// TwinCAT 3 PLC project EIOSM000003
// ProgramVersion: 3.1.4024.0
// libraries:
//   EfficientIO Communicator, * (EfficientIO)
//   EfficientIO Energy Basic, * (EfficientIO)
//   Lynus Persistent Data V1, * (Lynus AG)
//   Lynus Standards, * (EfficientIO)
//   Tc2_EtherCAT, * (Beckhoff Automation GmbH)
//   Tc2_Standard, * (Beckhoff Automation GmbH)
//   Tc2_System, * (Beckhoff Automation GmbH)
//   Tc2_Utilities, * (Beckhoff Automation GmbH)
//   Tc3_IPCDiag, * (Beckhoff Automation GmbH)
//   Tc3_Module, * (Beckhoff Automation GmbH)
// project tree:
//   ENUM/ E_State.TcDUT (not stored)
//   / FastTask.TcTTO, PlcTask.TcTTO, SlowTask.TcTTO
//   FBs/EL3443_DPM/DUTs/ E_EL3443_DPM_Phase.TcDUT (not stored), E_EL3443_DPM_Total.TcDUT (not stored), MDP5001_341_7CD731EE.TcDUT (not stored), MDP5001_341_I_7CD731EE.TcDUT (not stored), MDP5001_341_O_7CD731EE.TcDUT (not stored), ST_EL3443_DPM_MUX_REAL.TcDUT (not stored), ST_EL3443_DPM_MUX_ULINT.TcDUT (not stored), ST_EL3443_DPM_StatusLx.TcDUT (not stored), ST_EL3443_DPM_StatusTotal.TcDUT (not stored), ST_EL3443_DPM_VariantLx.TcDUT (not stored), ST_EL3443_DPM_VariantTotal.TcDUT (not stored), ST_EL3443_DPM_VariantValues.TcDUT (not stored)
//   FBs/EL3443_DPM/ FB_EL3443_DPM.TcPOU (not stored)
//   FBs/EL3446 FW02 or higher/DUTs/ E_EL3446_Phase.TcDUT (not stored), MDP5001_342_066CA8C6.TcDUT (not stored), MDP5001_342_I_066CA8C6.TcDUT (not stored), MDP5001_342_O_066CA8C6.TcDUT (not stored), ST_EL3446_MUX_REAL.TcDUT (not stored), ST_EL3446_MUX_ULINT.TcDUT (not stored), ST_EL3446_StatusIx.TcDUT (not stored), ST_EL3446_VariantIx.TcDUT (not stored), ST_EL3446_VariantValues.TcDUT (not stored)
//   FBs/EL3446 FW02 or higher/ FB_EL3446.TcPOU (not stored)
//   FBs/ FB_CoE_EL3443.TcPOU (not stored), FB_CoE_EL3446.TcPOU (not stored), FB_EM_Beckhoff_EL3443.TcPOU (not stored), FB_EM_Beckhoff_EL3446.TcPOU (not stored), FB_PT100_Read.TcPOU, prg_ReadDeviceName.TcPOU (not stored)
//   POUs/ prgComEffIO.TcPOU, prgEM.TcPOU, prgHW.TcPOU (not stored), prgPersistent.TcPOU (not stored), prgRWEffIO.TcPOU (not stored), prgTmp.TcPOU, prgVarEffIO.TcPOU (not stored)
// real-time tasks:
//   TASK MiddleTask: cycle T#10ms, priority 20, ADS port 350
//   TASK FastTask: cycle T#5ms, priority 19, ADS port 351
//   TASK SlowTask: cycle T#20ms, priority 21, ADS port 352
// I/O:
//   DEVICE Device 1 (Beckhoff CCAT)
//   DEVICE Device 2 (EtherCAT), AmsNetId 5.146.122.92.3.1
//     Term 1 (EK1200) [EK1200-5000 EtherCAT Power supply (2A E-Bus)]
//       Term 2 (EL3443) [EL3443 3Ch. Power Measuring]
//       Term 3 (EL3446) [EL3446 6 Ch.DPM Current Measurement Terminal]
//       Term 4 (EL3446) [EL3446 6 Ch.DPM Current Measurement Terminal]
//       Term 5 (EL3446) [EL3446 6 Ch.DPM Current Measurement Terminal]
//       Term 6 (EL3446) [EL3446 6 Ch.DPM Current Measurement Terminal]
//       Term 7 (EL3202) [EL3202 2Ch. Ana. Input PT100 (RTD)]
//       Term 8 (EL9011) [EL9011 End Terminal]
// variable links:
//   EIOSM000003/EIOSM000003 Instance <-> Device 2 (EtherCAT)/Term 1 (EK1200)/Term 2 (EL3443)
//     PlcTask Inputs/prgHW.MDP5001_341_DPM_Data_Data_{1..20} <-> DPM Data/Data {1..20}  (20 links)
//     PlcTask Inputs/prgHW.MDP5001_341_L1_Basic_Current <-> L1 Basic/Current
//     PlcTask Inputs/prgHW.MDP5001_341_L2_Basic_Current <-> L2 Basic/Current
//     PlcTask Inputs/prgHW.MDP5001_341_L3_Basic_Current <-> L3 Basic/Current
//     PlcTask Inputs/prgHW.MDP5001_341_L1_Basic_Voltage <-> L1 Basic/Voltage
//     PlcTask Inputs/prgHW.MDP5001_341_L2_Basic_Voltage <-> L2 Basic/Voltage
//     PlcTask Inputs/prgHW.MDP5001_341_L3_Basic_Voltage <-> L3 Basic/Voltage
//     PlcTask Inputs/prgHW.MDP5001_341_L1_Power_Active_Power <-> L1 Power/Active Power
//     PlcTask Inputs/prgHW.MDP5001_341_L2_Power_Active_Power <-> L2 Power/Active Power
//     PlcTask Inputs/prgHW.MDP5001_341_L3_Power_Active_Power <-> L3 Power/Active Power
//     PlcTask Inputs/prgHW.MDP5001_341_L1_Power_Apparent_Power <-> L1 Power/Apparent Power
//     PlcTask Inputs/prgHW.MDP5001_341_L2_Power_Apparent_Power <-> L2 Power/Apparent Power
//     PlcTask Inputs/prgHW.MDP5001_341_L3_Power_Apparent_Power <-> L3 Power/Apparent Power
//     PlcTask Inputs/prgHW.MDP5001_341_L1_Power_Power_Factor <-> L1 Power/Power Factor
//     PlcTask Inputs/prgHW.MDP5001_341_L2_Power_Power_Factor <-> L2 Power/Power Factor
//     PlcTask Inputs/prgHW.MDP5001_341_L3_Power_Power_Factor <-> L3 Power/Power Factor
//     PlcTask Inputs/prgHW.MDP5001_341_L1_Power_Reactive_Power <-> L1 Power/Reactive Power
//     PlcTask Inputs/prgHW.MDP5001_341_L2_Power_Reactive_Power <-> L2 Power/Reactive Power
//     PlcTask Inputs/prgHW.MDP5001_341_L3_Power_Reactive_Power <-> L3 Power/Reactive Power
//     PlcTask Inputs/prgHW.MDP5001_341_L1_Status_Current_Guard_Error <-> L1 Status/Current Guard Error
//     PlcTask Inputs/prgHW.MDP5001_341_L2_Status_Current_Guard_Error <-> L2 Status/Current Guard Error
//     PlcTask Inputs/prgHW.MDP5001_341_L3_Status_Current_Guard_Error <-> L3 Status/Current Guard Error
//     PlcTask Inputs/prgHW.MDP5001_341_L1_Status_Current_Guard_Warning <-> L1 Status/Current Guard Warning
//     PlcTask Inputs/prgHW.MDP5001_341_L2_Status_Current_Guard_Warning <-> L2 Status/Current Guard Warning
//     PlcTask Inputs/prgHW.MDP5001_341_L3_Status_Current_Guard_Warning <-> L3 Status/Current Guard Warning
//     PlcTask Inputs/prgHW.MDP5001_341_L1_Status_Inaccurate_Current <-> L1 Status/Inaccurate Current
//     PlcTask Inputs/prgHW.MDP5001_341_L2_Status_Inaccurate_Current <-> L2 Status/Inaccurate Current
//     PlcTask Inputs/prgHW.MDP5001_341_L3_Status_Inaccurate_Current <-> L3 Status/Inaccurate Current
//     PlcTask Inputs/prgHW.MDP5001_341_L1_Status_Inaccurate_Voltage <-> L1 Status/Inaccurate Voltage
//     PlcTask Inputs/prgHW.MDP5001_341_L2_Status_Inaccurate_Voltage <-> L2 Status/Inaccurate Voltage
//     PlcTask Inputs/prgHW.MDP5001_341_L3_Status_Inaccurate_Voltage <-> L3 Status/Inaccurate Voltage
//     PlcTask Inputs/prgHW.MDP5001_341_L1_Status_Overcurrent <-> L1 Status/Overcurrent
//     PlcTask Inputs/prgHW.MDP5001_341_L2_Status_Overcurrent <-> L2 Status/Overcurrent
//     PlcTask Inputs/prgHW.MDP5001_341_L3_Status_Overcurrent <-> L3 Status/Overcurrent
//     PlcTask Inputs/prgHW.MDP5001_341_L1_Status_Overvoltage <-> L1 Status/Overvoltage
//     PlcTask Inputs/prgHW.MDP5001_341_L2_Status_Overvoltage <-> L2 Status/Overvoltage
//     PlcTask Inputs/prgHW.MDP5001_341_L3_Status_Overvoltage <-> L3 Status/Overvoltage
//     PlcTask Inputs/prgHW.MDP5001_341_L1_Status_TxPDO_Toggle <-> L1 Status/TxPDO Toggle
//     PlcTask Inputs/prgHW.MDP5001_341_L2_Status_TxPDO_Toggle <-> L2 Status/TxPDO Toggle
//     PlcTask Inputs/prgHW.MDP5001_341_L3_Status_TxPDO_Toggle <-> L3 Status/TxPDO Toggle
//     PlcTask Inputs/prgHW.MDP5001_341_L1_Status_Voltage_Guard_Error <-> L1 Status/Voltage Guard Error
//     PlcTask Inputs/prgHW.MDP5001_341_L2_Status_Voltage_Guard_Error <-> L2 Status/Voltage Guard Error
//     PlcTask Inputs/prgHW.MDP5001_341_L3_Status_Voltage_Guard_Error <-> L3 Status/Voltage Guard Error
//     PlcTask Inputs/prgHW.MDP5001_341_L1_Status_Voltage_Guard_Warning <-> L1 Status/Voltage Guard Warning
//     PlcTask Inputs/prgHW.MDP5001_341_L2_Status_Voltage_Guard_Warning <-> L2 Status/Voltage Guard Warning
//     PlcTask Inputs/prgHW.MDP5001_341_L3_Status_Voltage_Guard_Warning <-> L3 Status/Voltage Guard Warning
//     PlcTask Inputs/prgHW.MDP5001_341_L1_Status_Voltage_Sign_Bit <-> L1 Status/Voltage Sign Bit
//     PlcTask Inputs/prgHW.MDP5001_341_L2_Status_Voltage_Sign_Bit <-> L2 Status/Voltage Sign Bit
//     PlcTask Inputs/prgHW.MDP5001_341_L3_Status_Voltage_Sign_Bit <-> L3 Status/Voltage Sign Bit
//     PlcTask Inputs/prgHW.MDP5001_341_Total_Basic_Calculated_Neutral_Line_Current <-> Total Basic/Calculated Neutral Line Current
//     PlcTask Inputs/prgHW.MDP5001_341_Total_Basic_Frequency <-> Total Basic/Frequency
//     PlcTask Inputs/prgHW.MDP5001_341_Total_Basic_Power_Factor <-> Total Basic/Power Factor
//     PlcTask Inputs/prgHW.MDP5001_341_Total_Status_Active_Power_Guard_Error <-> Total Status/Active Power Guard Error
//     PlcTask Inputs/prgHW.MDP5001_341_Total_Status_Active_Power_Guard_Warning <-> Total Status/Active Power Guard Warning
//     PlcTask Inputs/prgHW.MDP5001_341_Total_Status_Apparent_Power_Guard_Error <-> Total Status/Apparent Power Guard Error
//     PlcTask Inputs/prgHW.MDP5001_341_Total_Status_Apparent_Power_Guard_Warning <-> Total Status/Apparent Power Guard Warning
//     PlcTask Inputs/prgHW.MDP5001_341_Total_Status_Frequency_Guard_Error <-> Total Status/Frequency Guard Error
//     PlcTask Inputs/prgHW.MDP5001_341_Total_Status_Frequency_Guard_Warning <-> Total Status/Frequency Guard Warning
//     PlcTask Inputs/prgHW.MDP5001_341_Total_Status_Grid_Direction <-> Total Status/Grid Direction
//     PlcTask Inputs/prgHW.MDP5001_341_Total_Status_Neutral_Current_Guard_Error <-> Total Status/Neutral Current Guard Error
//     PlcTask Inputs/prgHW.MDP5001_341_Total_Status_Neutral_Current_Guard_Warning <-> Total Status/Neutral Current Guard Warning
//     PlcTask Inputs/prgHW.MDP5001_341_Total_Status_Power_Quality_Factor <-> Total Status/Power Quality Factor
//     PlcTask Inputs/prgHW.MDP5001_341_Total_Status_Power_Quality_Guard_Error <-> Total Status/Power Quality Guard Error
//     PlcTask Inputs/prgHW.MDP5001_341_Total_Status_Power_Quality_Guard_Warning <-> Total Status/Power Quality Guard Warning
//     PlcTask Inputs/prgHW.MDP5001_341_Total_Status_System_State <-> Total Status/System State
//     PlcTask Inputs/prgHW.MDP5001_341_Total_Status_TxPDO_State <-> Total Status/TxPDO State
//     PlcTask Inputs/prgHW.MDP5001_341_Total_Status_TxPDO_Toggle <-> Total Status/TxPDO Toggle
//     PlcTask Inputs/prgHW.MDP5001_341_Total_Variant_Value_In_Index_1_REAL <-> Total Variant Value In/Index 1 REAL
//     PlcTask Inputs/prgHW.MDP5001_341_Total_Variant_Value_In_Index_2_REAL <-> Total Variant Value In/Index 2 REAL
//     PlcTask Inputs/prgHW.MDP5001_341_Total_Variant_Value_In_Index_3_REAL <-> Total Variant Value In/Index 3 REAL
//     PlcTask Inputs/prgHW.MDP5001_341_Total_Variant_Value_In_Index_4_ULINT <-> Total Variant Value In/Index 4 ULINT
//     PlcTask Inputs/prgHW.MDP5001_341_Total_Variant_Value_In_TxPDO_Toggle <-> Total Variant Value In/TxPDO Toggle
//     PlcTask Inputs/prgHW.MDP5001_341_Total_Variant_Value_In_Value_1_REAL <-> Total Variant Value In/Value 1 REAL
//     PlcTask Inputs/prgHW.MDP5001_341_Total_Variant_Value_In_Value_2_REAL <-> Total Variant Value In/Value 2 REAL
//     PlcTask Inputs/prgHW.MDP5001_341_Total_Variant_Value_In_Value_3_REAL <-> Total Variant Value In/Value 3 REAL
//     PlcTask Inputs/prgHW.MDP5001_341_Total_Variant_Value_In_Value_4_ULINT <-> Total Variant Value In/Value 4 ULINT
//     PlcTask Outputs/prgHW.MDP5001_341_Total_Interval_Reset_Interval <-> Total Interval/Reset Interval
//     PlcTask Outputs/prgHW.MDP5001_341_Total_Variant_Value_Out_Index_1_REAL <-> Total Variant Value Out/Index 1 REAL
//     PlcTask Outputs/prgHW.MDP5001_341_Total_Variant_Value_Out_Index_2_REAL <-> Total Variant Value Out/Index 2 REAL
//     PlcTask Outputs/prgHW.MDP5001_341_Total_Variant_Value_Out_Index_3_REAL <-> Total Variant Value Out/Index 3 REAL
//     PlcTask Outputs/prgHW.MDP5001_341_Total_Variant_Value_Out_Index_4_ULINT <-> Total Variant Value Out/Index 4 ULINT
//   EIOSM000003/EIOSM000003 Instance <-> Device 2 (EtherCAT)/Term 1 (EK1200)/Term 3 (EL3446)
//     PlcTask Inputs/prgHW.MDP5001_342_DPM_Variant_Value_In_Index_1_REAL_EM1 <-> DPM Variant Value In/Index 1 REAL
//     PlcTask Inputs/prgHW.MDP5001_342_DPM_Variant_Value_In_Index_2_REAL_EM1 <-> DPM Variant Value In/Index 2 REAL
//     PlcTask Inputs/prgHW.MDP5001_342_DPM_Variant_Value_In_Index_3_REAL_EM1 <-> DPM Variant Value In/Index 3 REAL
//     PlcTask Inputs/prgHW.MDP5001_342_DPM_Variant_Value_In_Index_4_ULINT_EM1 <-> DPM Variant Value In/Index 4 ULINT
//     PlcTask Inputs/prgHW.MDP5001_342_DPM_Variant_Value_In_TxPDO_Toggle_EM1 <-> DPM Variant Value In/TxPDO Toggle
//     PlcTask Inputs/prgHW.MDP5001_342_DPM_Variant_Value_In_Value_1_REAL_EM1 <-> DPM Variant Value In/Value 1 REAL
//     PlcTask Inputs/prgHW.MDP5001_342_DPM_Variant_Value_In_Value_2_REAL_EM1 <-> DPM Variant Value In/Value 2 REAL
//     PlcTask Inputs/prgHW.MDP5001_342_DPM_Variant_Value_In_Value_3_REAL_EM1 <-> DPM Variant Value In/Value 3 REAL
//     PlcTask Inputs/prgHW.MDP5001_342_DPM_Variant_Value_In_Value_4_ULINT_EM1 <-> DPM Variant Value In/Value 4 ULINT
//     PlcTask Inputs/prgHW.MDP5001_342_I{1..6}_Channel_Active_Energy_EM1 <-> I{1..6} Channel/Active Energy  (6 links)
//     PlcTask Inputs/prgHW.MDP5001_342_I{1..6}_Channel_Active_Power_EM1 <-> I{1..6} Channel/Active Power  (6 links)
//     PlcTask Inputs/prgHW.MDP5001_342_I{1..6}_Channel_Active_Power_Guard_Error_EM1 <-> I{1..6} Channel/Active Power Guard Error  (6 links)
//     PlcTask Inputs/prgHW.MDP5001_342_I{1..6}_Channel_Active_Power_Guard_Warning_EM1 <-> I{1..6} Channel/Active Power Guard Warning  (6 links)
//     PlcTask Inputs/prgHW.MDP5001_342_I{1..6}_Channel_Apparent_Power_EM1 <-> I{1..6} Channel/Apparent Power  (6 links)
//     PlcTask Inputs/prgHW.MDP5001_342_I{1..6}_Channel_Apparent_Power_Guard_Error_EM1 <-> I{1..6} Channel/Apparent Power Guard Error  (6 links)
//     PlcTask Inputs/prgHW.MDP5001_342_I{1..6}_Channel_Apparent_Power_Guard_Warning_EM1 <-> I{1..6} Channel/Apparent Power Guard Warning  (6 links)
//     PlcTask Inputs/prgHW.MDP5001_342_I{1..6}_Channel_Current_EM1 <-> I{1..6} Channel/Current  (6 links)
//     PlcTask Inputs/prgHW.MDP5001_342_I{1..6}_Channel_Current_Guard_Error_EM1 <-> I{1..6} Channel/Current Guard Error  (6 links)
//     PlcTask Inputs/prgHW.MDP5001_342_I{1..6}_Channel_Current_Guard_Warning_EM1 <-> I{1..6} Channel/Current Guard Warning  (6 links)
//     PlcTask Inputs/prgHW.MDP5001_342_I{1..6}_Channel_DPM_Inaccurate_EM1 <-> I{1..6} Channel/DPM Inaccurate  (6 links)
//     PlcTask Inputs/prgHW.MDP5001_342_I{1..6}_Channel_DPM_Timeout_EM1 <-> I{1..6} Channel/DPM Timeout  (6 links)
//     PlcTask Inputs/prgHW.MDP5001_342_I{1..6}_Channel_Inaccurate_Current_EM1 <-> I{1..6} Channel/Inaccurate Current  (6 links)
//     PlcTask Inputs/prgHW.MDP5001_342_I{1..6}_Channel_Overcurrent_EM1 <-> I{1..6} Channel/Overcurrent  (6 links)
//     PlcTask Inputs/prgHW.MDP5001_342_I{1..6}_Channel_Reactive_Power_Fundamental_EM1 <-> I{1..6} Channel/Reactive Power Fundamental  (6 links)
//     PlcTask Inputs/prgHW.MDP5001_342_I{1..6}_Channel_Reactive_Power_Guard_Error_EM1 <-> I{1..6} Channel/Reactive Power Guard Error  (6 links)
//     PlcTask Inputs/prgHW.MDP5001_342_I{1..6}_Channel_Reactive_Power_Guard_Warning_EM1 <-> I{1..6} Channel/Reactive Power Guard Warning  (6 links)
//     PlcTask Inputs/prgHW.MDP5001_342_I{1..6}_Channel_TxPDO_Toggle_EM1 <-> I{1..6} Channel/TxPDO Toggle  (6 links)
//     PlcTask Outputs/prgHW.MDP5001_342_DPM_Data_Data_{1..20}_EM1 <-> DPM Data/Data {1..20}  (20 links)
//     PlcTask Outputs/prgHW.MDP5001_342_DPM_Variant_Value_Out_Index_1_REAL_EM1 <-> DPM Variant Value Out/Index 1 REAL
//     PlcTask Outputs/prgHW.MDP5001_342_DPM_Variant_Value_Out_Index_2_REAL_EM1 <-> DPM Variant Value Out/Index 2 REAL
//     PlcTask Outputs/prgHW.MDP5001_342_DPM_Variant_Value_Out_Index_3_REAL_EM1 <-> DPM Variant Value Out/Index 3 REAL
//     PlcTask Outputs/prgHW.MDP5001_342_DPM_Variant_Value_Out_Index_4_ULINT_EM1 <-> DPM Variant Value Out/Index 4 ULINT
//   EIOSM000003/EIOSM000003 Instance <-> Device 2 (EtherCAT)/Term 1 (EK1200)/Term 4 (EL3446)
//     PlcTask Inputs/prgHW.MDP5001_342_DPM_Variant_Value_In_Index_1_REAL_EM2 <-> DPM Variant Value In/Index 1 REAL
//     PlcTask Inputs/prgHW.MDP5001_342_DPM_Variant_Value_In_Index_2_REAL_EM2 <-> DPM Variant Value In/Index 2 REAL
//     PlcTask Inputs/prgHW.MDP5001_342_DPM_Variant_Value_In_Index_3_REAL_EM2 <-> DPM Variant Value In/Index 3 REAL
//     PlcTask Inputs/prgHW.MDP5001_342_DPM_Variant_Value_In_Index_4_ULINT_EM2 <-> DPM Variant Value In/Index 4 ULINT
//     PlcTask Inputs/prgHW.MDP5001_342_DPM_Variant_Value_In_TxPDO_Toggle_EM2 <-> DPM Variant Value In/TxPDO Toggle
//     PlcTask Inputs/prgHW.MDP5001_342_DPM_Variant_Value_In_Value_1_REAL_EM2 <-> DPM Variant Value In/Value 1 REAL
//     PlcTask Inputs/prgHW.MDP5001_342_DPM_Variant_Value_In_Value_2_REAL_EM2 <-> DPM Variant Value In/Value 2 REAL
//     PlcTask Inputs/prgHW.MDP5001_342_DPM_Variant_Value_In_Value_3_REAL_EM2 <-> DPM Variant Value In/Value 3 REAL
//     PlcTask Inputs/prgHW.MDP5001_342_DPM_Variant_Value_In_Value_4_ULINT_EM2 <-> DPM Variant Value In/Value 4 ULINT
//     PlcTask Inputs/prgHW.MDP5001_342_I{1..6}_Channel_Active_Energy_EM2 <-> I{1..6} Channel/Active Energy  (6 links)
//     PlcTask Inputs/prgHW.MDP5001_342_I{1..6}_Channel_Active_Power_EM2 <-> I{1..6} Channel/Active Power  (6 links)
//     PlcTask Inputs/prgHW.MDP5001_342_I{1..6}_Channel_Active_Power_Guard_Error_EM2 <-> I{1..6} Channel/Active Power Guard Error  (6 links)
//     PlcTask Inputs/prgHW.MDP5001_342_I{1..6}_Channel_Active_Power_Guard_Warning_EM2 <-> I{1..6} Channel/Active Power Guard Warning  (6 links)
//     PlcTask Inputs/prgHW.MDP5001_342_I{1..6}_Channel_Apparent_Power_EM2 <-> I{1..6} Channel/Apparent Power  (6 links)
//     PlcTask Inputs/prgHW.MDP5001_342_I{1..6}_Channel_Apparent_Power_Guard_Error_EM2 <-> I{1..6} Channel/Apparent Power Guard Error  (6 links)
//     PlcTask Inputs/prgHW.MDP5001_342_I{1..6}_Channel_Apparent_Power_Guard_Warning_EM2 <-> I{1..6} Channel/Apparent Power Guard Warning  (6 links)
//     PlcTask Inputs/prgHW.MDP5001_342_I{1..6}_Channel_Current_EM2 <-> I{1..6} Channel/Current  (6 links)
//     PlcTask Inputs/prgHW.MDP5001_342_I{1..6}_Channel_Current_Guard_Error_EM2 <-> I{1..6} Channel/Current Guard Error  (6 links)
//     PlcTask Inputs/prgHW.MDP5001_342_I{1..6}_Channel_Current_Guard_Warning_EM2 <-> I{1..6} Channel/Current Guard Warning  (6 links)
//     PlcTask Inputs/prgHW.MDP5001_342_I{1..6}_Channel_DPM_Inaccurate_EM2 <-> I{1..6} Channel/DPM Inaccurate  (6 links)
//     PlcTask Inputs/prgHW.MDP5001_342_I{1..6}_Channel_DPM_Timeout_EM2 <-> I{1..6} Channel/DPM Timeout  (6 links)
//     PlcTask Inputs/prgHW.MDP5001_342_I{1..6}_Channel_Inaccurate_Current_EM2 <-> I{1..6} Channel/Inaccurate Current  (6 links)
//     PlcTask Inputs/prgHW.MDP5001_342_I{1..6}_Channel_Overcurrent_EM2 <-> I{1..6} Channel/Overcurrent  (6 links)
//     PlcTask Inputs/prgHW.MDP5001_342_I{1..6}_Channel_Reactive_Power_Fundamental_EM2 <-> I{1..6} Channel/Reactive Power Fundamental  (6 links)
//     PlcTask Inputs/prgHW.MDP5001_342_I{1..6}_Channel_Reactive_Power_Guard_Error_EM2 <-> I{1..6} Channel/Reactive Power Guard Error  (6 links)
//     PlcTask Inputs/prgHW.MDP5001_342_I{1..6}_Channel_Reactive_Power_Guard_Warning_EM2 <-> I{1..6} Channel/Reactive Power Guard Warning  (6 links)
//     PlcTask Inputs/prgHW.MDP5001_342_I{1..6}_Channel_TxPDO_Toggle_EM2 <-> I{1..6} Channel/TxPDO Toggle  (6 links)
//     PlcTask Outputs/prgHW.MDP5001_342_DPM_Data_Data_{1..20}_EM2 <-> DPM Data/Data {1..20}  (20 links)
//     PlcTask Outputs/prgHW.MDP5001_342_DPM_Variant_Value_Out_Index_1_REAL_EM2 <-> DPM Variant Value Out/Index 1 REAL
//     PlcTask Outputs/prgHW.MDP5001_342_DPM_Variant_Value_Out_Index_2_REAL_EM2 <-> DPM Variant Value Out/Index 2 REAL
//     PlcTask Outputs/prgHW.MDP5001_342_DPM_Variant_Value_Out_Index_3_REAL_EM2 <-> DPM Variant Value Out/Index 3 REAL
//     PlcTask Outputs/prgHW.MDP5001_342_DPM_Variant_Value_Out_Index_4_ULINT_EM2 <-> DPM Variant Value Out/Index 4 ULINT
//   EIOSM000003/EIOSM000003 Instance <-> Device 2 (EtherCAT)/Term 1 (EK1200)/Term 5 (EL3446)
//     PlcTask Inputs/prgHW.MDP5001_342_DPM_Variant_Value_In_Index_1_REAL_EM3 <-> DPM Variant Value In/Index 1 REAL
//     PlcTask Inputs/prgHW.MDP5001_342_DPM_Variant_Value_In_Index_2_REAL_EM3 <-> DPM Variant Value In/Index 2 REAL
//     PlcTask Inputs/prgHW.MDP5001_342_DPM_Variant_Value_In_Index_3_REAL_EM3 <-> DPM Variant Value In/Index 3 REAL
//     PlcTask Inputs/prgHW.MDP5001_342_DPM_Variant_Value_In_Index_4_ULINT_EM3 <-> DPM Variant Value In/Index 4 ULINT
//     PlcTask Inputs/prgHW.MDP5001_342_DPM_Variant_Value_In_TxPDO_Toggle_EM3 <-> DPM Variant Value In/TxPDO Toggle
//     PlcTask Inputs/prgHW.MDP5001_342_DPM_Variant_Value_In_Value_1_REAL_EM3 <-> DPM Variant Value In/Value 1 REAL
//     PlcTask Inputs/prgHW.MDP5001_342_DPM_Variant_Value_In_Value_2_REAL_EM3 <-> DPM Variant Value In/Value 2 REAL
//     PlcTask Inputs/prgHW.MDP5001_342_DPM_Variant_Value_In_Value_3_REAL_EM3 <-> DPM Variant Value In/Value 3 REAL
//     PlcTask Inputs/prgHW.MDP5001_342_DPM_Variant_Value_In_Value_4_ULINT_EM3 <-> DPM Variant Value In/Value 4 ULINT
//     PlcTask Inputs/prgHW.MDP5001_342_I{1..6}_Channel_Active_Energy_EM3 <-> I{1..6} Channel/Active Energy  (6 links)
//     PlcTask Inputs/prgHW.MDP5001_342_I{1..6}_Channel_Active_Power_EM3 <-> I{1..6} Channel/Active Power  (6 links)
//     PlcTask Inputs/prgHW.MDP5001_342_I{1..6}_Channel_Active_Power_Guard_Error_EM3 <-> I{1..6} Channel/Active Power Guard Error  (6 links)
//     PlcTask Inputs/prgHW.MDP5001_342_I{1..6}_Channel_Active_Power_Guard_Warning_EM3 <-> I{1..6} Channel/Active Power Guard Warning  (6 links)
//     PlcTask Inputs/prgHW.MDP5001_342_I{1..6}_Channel_Apparent_Power_EM3 <-> I{1..6} Channel/Apparent Power  (6 links)
//     PlcTask Inputs/prgHW.MDP5001_342_I{1..6}_Channel_Apparent_Power_Guard_Error_EM3 <-> I{1..6} Channel/Apparent Power Guard Error  (6 links)
//     PlcTask Inputs/prgHW.MDP5001_342_I{1..6}_Channel_Apparent_Power_Guard_Warning_EM3 <-> I{1..6} Channel/Apparent Power Guard Warning  (6 links)
//     PlcTask Inputs/prgHW.MDP5001_342_I{1..6}_Channel_Current_EM3 <-> I{1..6} Channel/Current  (6 links)
//     PlcTask Inputs/prgHW.MDP5001_342_I{1..6}_Channel_Current_Guard_Error_EM3 <-> I{1..6} Channel/Current Guard Error  (6 links)
//     PlcTask Inputs/prgHW.MDP5001_342_I{1..6}_Channel_Current_Guard_Warning_EM3 <-> I{1..6} Channel/Current Guard Warning  (6 links)
//     PlcTask Inputs/prgHW.MDP5001_342_I{1..6}_Channel_DPM_Inaccurate_EM3 <-> I{1..6} Channel/DPM Inaccurate  (6 links)
//     PlcTask Inputs/prgHW.MDP5001_342_I{1..6}_Channel_DPM_Timeout_EM3 <-> I{1..6} Channel/DPM Timeout  (6 links)
//     PlcTask Inputs/prgHW.MDP5001_342_I{1..6}_Channel_Inaccurate_Current_EM3 <-> I{1..6} Channel/Inaccurate Current  (6 links)
//     PlcTask Inputs/prgHW.MDP5001_342_I{1..6}_Channel_Overcurrent_EM3 <-> I{1..6} Channel/Overcurrent  (6 links)
//     PlcTask Inputs/prgHW.MDP5001_342_I{1..6}_Channel_Reactive_Power_Fundamental_EM3 <-> I{1..6} Channel/Reactive Power Fundamental  (6 links)
//     PlcTask Inputs/prgHW.MDP5001_342_I{1..6}_Channel_Reactive_Power_Guard_Error_EM3 <-> I{1..6} Channel/Reactive Power Guard Error  (6 links)
//     PlcTask Inputs/prgHW.MDP5001_342_I{1..6}_Channel_Reactive_Power_Guard_Warning_EM3 <-> I{1..6} Channel/Reactive Power Guard Warning  (6 links)
//     PlcTask Inputs/prgHW.MDP5001_342_I{1..6}_Channel_TxPDO_Toggle_EM3 <-> I{1..6} Channel/TxPDO Toggle  (6 links)
//     PlcTask Outputs/prgHW.MDP5001_342_DPM_Data_Data_{1..20}_EM3 <-> DPM Data/Data {1..20}  (20 links)
//     PlcTask Outputs/prgHW.MDP5001_342_DPM_Variant_Value_Out_Index_1_REAL_EM3 <-> DPM Variant Value Out/Index 1 REAL
//     PlcTask Outputs/prgHW.MDP5001_342_DPM_Variant_Value_Out_Index_2_REAL_EM3 <-> DPM Variant Value Out/Index 2 REAL
//     PlcTask Outputs/prgHW.MDP5001_342_DPM_Variant_Value_Out_Index_3_REAL_EM3 <-> DPM Variant Value Out/Index 3 REAL
//     PlcTask Outputs/prgHW.MDP5001_342_DPM_Variant_Value_Out_Index_4_ULINT_EM3 <-> DPM Variant Value Out/Index 4 ULINT
//   EIOSM000003/EIOSM000003 Instance <-> Device 2 (EtherCAT)/Term 1 (EK1200)/Term 6 (EL3446)
//     PlcTask Inputs/prgHW.MDP5001_342_DPM_Variant_Value_In_Index_1_REAL_EM4 <-> DPM Variant Value In/Index 1 REAL
//     PlcTask Inputs/prgHW.MDP5001_342_DPM_Variant_Value_In_Index_2_REAL_EM4 <-> DPM Variant Value In/Index 2 REAL
//     PlcTask Inputs/prgHW.MDP5001_342_DPM_Variant_Value_In_Index_3_REAL_EM4 <-> DPM Variant Value In/Index 3 REAL
//     PlcTask Inputs/prgHW.MDP5001_342_DPM_Variant_Value_In_Index_4_ULINT_EM4 <-> DPM Variant Value In/Index 4 ULINT
//     PlcTask Inputs/prgHW.MDP5001_342_DPM_Variant_Value_In_TxPDO_Toggle_EM4 <-> DPM Variant Value In/TxPDO Toggle
//     PlcTask Inputs/prgHW.MDP5001_342_DPM_Variant_Value_In_Value_1_REAL_EM4 <-> DPM Variant Value In/Value 1 REAL
//     PlcTask Inputs/prgHW.MDP5001_342_DPM_Variant_Value_In_Value_2_REAL_EM4 <-> DPM Variant Value In/Value 2 REAL
//     PlcTask Inputs/prgHW.MDP5001_342_DPM_Variant_Value_In_Value_3_REAL_EM4 <-> DPM Variant Value In/Value 3 REAL
//     PlcTask Inputs/prgHW.MDP5001_342_DPM_Variant_Value_In_Value_4_ULINT_EM4 <-> DPM Variant Value In/Value 4 ULINT
//     PlcTask Inputs/prgHW.MDP5001_342_I{1..6}_Channel_Active_Energy_EM4 <-> I{1..6} Channel/Active Energy  (6 links)
//     PlcTask Inputs/prgHW.MDP5001_342_I{1..6}_Channel_Active_Power_EM4 <-> I{1..6} Channel/Active Power  (6 links)
//     PlcTask Inputs/prgHW.MDP5001_342_I{1..6}_Channel_Active_Power_Guard_Error_EM4 <-> I{1..6} Channel/Active Power Guard Error  (6 links)
//     PlcTask Inputs/prgHW.MDP5001_342_I{1..6}_Channel_Active_Power_Guard_Warning_EM4 <-> I{1..6} Channel/Active Power Guard Warning  (6 links)
//     PlcTask Inputs/prgHW.MDP5001_342_I{1..6}_Channel_Apparent_Power_EM4 <-> I{1..6} Channel/Apparent Power  (6 links)
//     PlcTask Inputs/prgHW.MDP5001_342_I{1..6}_Channel_Apparent_Power_Guard_Error_EM4 <-> I{1..6} Channel/Apparent Power Guard Error  (6 links)
//     PlcTask Inputs/prgHW.MDP5001_342_I{1..6}_Channel_Apparent_Power_Guard_Warning_EM4 <-> I{1..6} Channel/Apparent Power Guard Warning  (6 links)
//     PlcTask Inputs/prgHW.MDP5001_342_I{1..6}_Channel_Current_EM4 <-> I{1..6} Channel/Current  (6 links)
//     PlcTask Inputs/prgHW.MDP5001_342_I{1..6}_Channel_Current_Guard_Error_EM4 <-> I{1..6} Channel/Current Guard Error  (6 links)
//     PlcTask Inputs/prgHW.MDP5001_342_I{1..6}_Channel_Current_Guard_Warning_EM4 <-> I{1..6} Channel/Current Guard Warning  (6 links)
//     PlcTask Inputs/prgHW.MDP5001_342_I{1..6}_Channel_DPM_Inaccurate_EM4 <-> I{1..6} Channel/DPM Inaccurate  (6 links)
//     PlcTask Inputs/prgHW.MDP5001_342_I{1..6}_Channel_DPM_Timeout_EM4 <-> I{1..6} Channel/DPM Timeout  (6 links)
//     PlcTask Inputs/prgHW.MDP5001_342_I{1..6}_Channel_Inaccurate_Current_EM4 <-> I{1..6} Channel/Inaccurate Current  (6 links)
//     PlcTask Inputs/prgHW.MDP5001_342_I{1..6}_Channel_Overcurrent_EM4 <-> I{1..6} Channel/Overcurrent  (6 links)
//     PlcTask Inputs/prgHW.MDP5001_342_I{1..6}_Channel_Reactive_Power_Fundamental_EM4 <-> I{1..6} Channel/Reactive Power Fundamental  (6 links)
//     PlcTask Inputs/prgHW.MDP5001_342_I{1..6}_Channel_Reactive_Power_Guard_Error_EM4 <-> I{1..6} Channel/Reactive Power Guard Error  (6 links)
//     PlcTask Inputs/prgHW.MDP5001_342_I{1..6}_Channel_Reactive_Power_Guard_Warning_EM4 <-> I{1..6} Channel/Reactive Power Guard Warning  (6 links)
//     PlcTask Inputs/prgHW.MDP5001_342_I{1..6}_Channel_TxPDO_Toggle_EM4 <-> I{1..6} Channel/TxPDO Toggle  (6 links)
//     PlcTask Outputs/prgHW.MDP5001_342_DPM_Data_Data_{1..20}_EM4 <-> DPM Data/Data {1..20}  (20 links)
//     PlcTask Outputs/prgHW.MDP5001_342_DPM_Variant_Value_Out_Index_1_REAL_EM4 <-> DPM Variant Value Out/Index 1 REAL
//     PlcTask Outputs/prgHW.MDP5001_342_DPM_Variant_Value_Out_Index_2_REAL_EM4 <-> DPM Variant Value Out/Index 2 REAL
//     PlcTask Outputs/prgHW.MDP5001_342_DPM_Variant_Value_Out_Index_3_REAL_EM4 <-> DPM Variant Value Out/Index 3 REAL
//     PlcTask Outputs/prgHW.MDP5001_342_DPM_Variant_Value_Out_Index_4_ULINT_EM4 <-> DPM Variant Value Out/Index 4 ULINT
//   EIOSM000003/EIOSM000003 Instance <-> Device 2 (EtherCAT)/Term 1 (EK1200)/Term 7 (EL3202)
//     PlcTask Inputs/prgTmp.EL3202_Channel_1 <-> RTD Inputs Channel 1/Value
//     PlcTask Inputs/prgTmp.EL3202_Channel_2 <-> RTD Inputs Channel 2/Value

CONFIGURATION EIOSM000003
    RESOURCE PLC ON TwinCAT3
        TASK FastTask(INTERVAL := T#5ms, PRIORITY := 19);
        TASK PlcTask(INTERVAL := T#10ms, PRIORITY := 20);
        TASK SlowTask(INTERVAL := T#20ms, PRIORITY := 21);
        PROGRAM prgVarEffIO WITH FastTask : prgVarEffIO;
        PROGRAM prgRWEffIO WITH FastTask : prgRWEffIO;
        PROGRAM prgPersistent WITH FastTask : prgPersistent;
        PROGRAM prgHW WITH PlcTask : prgHW;
        PROGRAM prgEM WITH PlcTask : prgEM;
        PROGRAM prgTmp WITH PlcTask : prgTmp;
        PROGRAM prgComEffIO WITH SlowTask : prgComEffIO;
    END_RESOURCE
END_CONFIGURATION

// ---- POUs/prgEM.TcPOU
PROGRAM prgEM
VAR
 	fb_EL3443_EM0 		: FB_EM_Beckhoff_EL3443;
	fb_EL3446_1			: FB_EM_Beckhoff_EL3446;
	fb_EL3446_2			: FB_EM_Beckhoff_EL3446;
	fb_EL3446_3			: FB_EM_Beckhoff_EL3446;
	fb_EL3446_4			: FB_EM_Beckhoff_EL3446;
	
	//EM0 (CEE32 3phase Measurement, EL3443)
	lr_RealPower_EM0		: LREAL;					//{#lynus.ag#()}
	lr_ApparentPower_EM0	: LREAL;					//{#lynus.ag#()}
	lr_ReactivePower_EM0	: LREAL;					//{#lynus.ag#()}
	lr_Frequency_EM0		: LREAL;					//{#lynus.ag#()}
	lr_Voltage_EM0_L1N		: LREAL;					//{#lynus.ag#()}
	lr_Voltage_EM0_L2N		: LREAL;					//{#lynus.ag#()}
	lr_Voltage_EM0_L3N		: LREAL;					//{#lynus.ag#()}
	lr_Voltage_EM0_L1L2		: LREAL;					//{#lynus.ag#()}
	lr_Voltage_EM0_L2L3		: LREAL;					//{#lynus.ag#()}
	lr_Voltage_EM0_L3L1		: LREAL;					//{#lynus.ag#()}
 	lr_Current_EM0_L1		: LREAL;					//{#lynus.ag#()}
	lr_Current_EM0_L2		: LREAL;					//{#lynus.ag#()}
	lr_Current_EM0_L3		: LREAL;					//{#lynus.ag#()}
	
	//EM1, EL3446-1
	lrPower_EM1_1		: LREAL;						//{#lynus.ag#()}
	lrPower_EM1_2		: LREAL;						//{#lynus.ag#()}
	lrPower_EM1_3		: LREAL;						//{#lynus.ag#()}
	lrPower_EM1_4		: LREAL;						//{#lynus.ag#()}
	lrPower_EM1_5		: LREAL;						//{#lynus.ag#()}
	lrPower_EM1_6		: LREAL;						//{#lynus.ag#()}
	lrPower_EM1_3p1		: LREAL;						//{#lynus.ag#()}
	lrPower_EM1_3p2		: LREAL;						//{#lynus.ag#()}
	
	//EM2, EL3446-2
	lrPower_EM2_1		: LREAL;						//{#lynus.ag#()}
	lrPower_EM2_2		: LREAL;						//{#lynus.ag#()}
	lrPower_EM2_3		: LREAL;						//{#lynus.ag#()}
	lrPower_EM2_4		: LREAL;						//{#lynus.ag#()}
	lrPower_EM2_5		: LREAL;						//{#lynus.ag#()}
	lrPower_EM2_6		: LREAL;						//{#lynus.ag#()}
	lrPower_EM2_3p1		: LREAL;						//{#lynus.ag#()}
	lrPower_EM2_3p2		: LREAL;						//{#lynus.ag#()}
	
	//EM3, EL3446-3
	lrPower_EM3_1		: LREAL;						//{#lynus.ag#()}
	lrPower_EM3_2		: LREAL;						//{#lynus.ag#()}
	lrPower_EM3_3		: LREAL;						//{#lynus.ag#()}
	lrPower_EM3_4		: LREAL;						//{#lynus.ag#()}
	lrPower_EM3_5		: LREAL;						//{#lynus.ag#()}
	lrPower_EM3_6		: LREAL;						//{#lynus.ag#()}
	lrPower_EM3_3p1		: LREAL;						//{#lynus.ag#()}
	lrPower_EM3_3p2		: LREAL;						//{#lynus.ag#()}
	
	//EM3, EL3446-4
	lrPower_EM4_1		: LREAL;						//{#lynus.ag#()}
	lrPower_EM4_2		: LREAL;						//{#lynus.ag#()}
	lrPower_EM4_3		: LREAL;						//{#lynus.ag#()}
	lrPower_EM4_4		: LREAL;						//{#lynus.ag#()}
	lrPower_EM4_5		: LREAL;						//{#lynus.ag#()}
	lrPower_EM4_6		: LREAL;						//{#lynus.ag#()}
	lrPower_EM4_3p1		: LREAL;						//{#lynus.ag#()}
	lrPower_EM4_3p2		: LREAL;						//{#lynus.ag#()}

END_VAR

VAR_INPUT
	stEL3443_IO_1 						: MDP5001_341_7CD731EE;
	stEL3446_IO_1 						: MDP5001_342_066CA8C6; 
	stEL3446_IO_2 						: MDP5001_342_066CA8C6;	
	stEL3446_IO_3 						: MDP5001_342_066CA8C6;	
	stEL3446_IO_4 						: MDP5001_342_066CA8C6;	
END_VAR

VAR PERSISTENT
	uiCurrentTransformerRatio_EM0	:UINT:=35;
	
	lr_EnergyCounter_EM0	: LREAL;
	lr_EnergyCounter_EM1	: LREAL;
	
	ui_PhaseSelector_EM1_1 : UINT := 1;						//{#lynus.ag#()}
	ui_PhaseSelector_EM1_2 : UINT := 2;						//{#lynus.ag#()}
	ui_PhaseSelector_EM1_3 : UINT := 3;						//{#lynus.ag#()}
	ui_PhaseSelector_EM1_4 : UINT := 1;						//{#lynus.ag#()}
	ui_PhaseSelector_EM1_5 : UINT := 2;						//{#lynus.ag#()}
	ui_PhaseSelector_EM1_6 : UINT := 3;						//{#lynus.ag#()}
	ui_PhaseSelector_EM2_1 : UINT := 1;						//{#lynus.ag#()}
	ui_PhaseSelector_EM2_2 : UINT := 2;						//{#lynus.ag#()}
	ui_PhaseSelector_EM2_3 : UINT := 3;						//{#lynus.ag#()}
	ui_PhaseSelector_EM2_4 : UINT := 1;						//{#lynus.ag#()}
	ui_PhaseSelector_EM2_5 : UINT := 2;						//{#lynus.ag#()}
	ui_PhaseSelector_EM2_6 : UINT := 3;						//{#lynus.ag#()}
	ui_PhaseSelector_EM3_1 : UINT := 1;						//{#lynus.ag#()}
	ui_PhaseSelector_EM3_2 : UINT := 2;						//{#lynus.ag#()}
	ui_PhaseSelector_EM3_3 : UINT := 3;						//{#lynus.ag#()}
	ui_PhaseSelector_EM3_4 : UINT := 1;						//{#lynus.ag#()}
	ui_PhaseSelector_EM3_5 : UINT := 2;						//{#lynus.ag#()}
	ui_PhaseSelector_EM3_6 : UINT := 3;						//{#lynus.ag#()}
	ui_PhaseSelector_EM4_1 : UINT := 1;						//{#lynus.ag#()}
	ui_PhaseSelector_EM4_2 : UINT := 2;						//{#lynus.ag#()}
	ui_PhaseSelector_EM4_3 : UINT := 3;						//{#lynus.ag#()}
	ui_PhaseSelector_EM4_4 : UINT := 1;						//{#lynus.ag#()}
	ui_PhaseSelector_EM4_5 : UINT := 2;						//{#lynus.ag#()}
	ui_PhaseSelector_EM4_6 : UINT := 3;						//{#lynus.ag#()}
	
	uiCurrentTransformerRatio_EM1_1	: UINT := 250;				//{#lynus.ag#()}
	uiCurrentTransformerRatio_EM1_2	: UINT := 250;				//{#lynus.ag#()}
	uiCurrentTransformerRatio_EM1_3	: UINT := 250;				//{#lynus.ag#()}
	uiCurrentTransformerRatio_EM1_4	: UINT := 35;				//{#lynus.ag#()}
	uiCurrentTransformerRatio_EM1_5	: UINT := 35;				//{#lynus.ag#()}
	uiCurrentTransformerRatio_EM1_6	: UINT := 35;				//{#lynus.ag#()}
	uiCurrentTransformerRatio_EM2_1	: UINT := 35;				//{#lynus.ag#()}
	uiCurrentTransformerRatio_EM2_2	: UINT := 35;				//{#lynus.ag#()}
	uiCurrentTransformerRatio_EM2_3	: UINT := 35;				//{#lynus.ag#()}
	uiCurrentTransformerRatio_EM2_4	: UINT := 35;				//{#lynus.ag#()}
	uiCurrentTransformerRatio_EM2_5	: UINT := 35;				//{#lynus.ag#()}
	uiCurrentTransformerRatio_EM2_6	: UINT := 35;				//{#lynus.ag#()}
	uiCurrentTransformerRatio_EM3_1	: UINT := 35;				//{#lynus.ag#()}
	uiCurrentTransformerRatio_EM3_2	: UINT := 35;				//{#lynus.ag#()}
	uiCurrentTransformerRatio_EM3_3	: UINT := 35;				//{#lynus.ag#()}
	uiCurrentTransformerRatio_EM3_4	: UINT := 35;				//{#lynus.ag#()}
	uiCurrentTransformerRatio_EM3_5	: UINT := 35;				//{#lynus.ag#()}
	uiCurrentTransformerRatio_EM3_6	: UINT := 35;				//{#lynus.ag#()}
	uiCurrentTransformerRatio_EM4_1	: UINT := 35;				//{#lynus.ag#()}
	uiCurrentTransformerRatio_EM4_2	: UINT := 35;				//{#lynus.ag#()}
	uiCurrentTransformerRatio_EM4_3	: UINT := 35;				//{#lynus.ag#()}
	uiCurrentTransformerRatio_EM4_4	: UINT := 35;				//{#lynus.ag#()}
	uiCurrentTransformerRatio_EM4_5	: UINT := 35;				//{#lynus.ag#()}
	uiCurrentTransformerRatio_EM4_6	: UINT := 35;				//{#lynus.ag#()}
	
	b_Invers_EM1_1	:	BOOL := FALSE;							//{#lynus.ag#()}
	b_Invers_EM1_2	:	BOOL := FALSE;							//{#lynus.ag#()}
	b_Invers_EM1_3	:	BOOL := FALSE;							//{#lynus.ag#()}
	b_Invers_EM1_4	:	BOOL := FALSE;							//{#lynus.ag#()}
	b_Invers_EM1_5	:	BOOL := FALSE;							//{#lynus.ag#()}
	b_Invers_EM1_6	:	BOOL := FALSE;							//{#lynus.ag#()}
	b_Invers_EM2_1	:	BOOL := FALSE;							//{#lynus.ag#()}
	b_Invers_EM2_2	:	BOOL := FALSE;							//{#lynus.ag#()}
	b_Invers_EM2_3	:	BOOL := FALSE;							//{#lynus.ag#()}
	b_Invers_EM2_4	:	BOOL := FALSE;							//{#lynus.ag#()}
	b_Invers_EM2_5	:	BOOL := FALSE;							//{#lynus.ag#()}
	b_Invers_EM2_6	:	BOOL := FALSE;							//{#lynus.ag#()}
	b_Invers_EM3_1	:	BOOL := FALSE;							//{#lynus.ag#()}
	b_Invers_EM3_2	:	BOOL := FALSE;							//{#lynus.ag#()}
	b_Invers_EM3_3	:	BOOL := FALSE;							//{#lynus.ag#()}
	b_Invers_EM3_4	:	BOOL := FALSE;							//{#lynus.ag#()}
	b_Invers_EM3_5	:	BOOL := FALSE;							//{#lynus.ag#()}
	b_Invers_EM3_6	:	BOOL := FALSE;							//{#lynus.ag#()}
	b_Invers_EM4_1	:	BOOL := FALSE;							//{#lynus.ag#()}
	b_Invers_EM4_2	:	BOOL := FALSE;							//{#lynus.ag#()}
	b_Invers_EM4_3	:	BOOL := FALSE;							//{#lynus.ag#()}
	b_Invers_EM4_4	:	BOOL := FALSE;							//{#lynus.ag#()}
	b_Invers_EM4_5	:	BOOL := FALSE;							//{#lynus.ag#()}
	b_Invers_EM4_6	:	BOOL := FALSE;							//{#lynus.ag#()}
END_VAR

//EM0 (CEE32 3phase Measurement)
fb_EL3443_EM0(
	bEnable 	:= TRUE, 
	bInvers_CH1 := , 
	bInvers_CH2	:= , 
	bInvers_CH3	:= , 
	uiCurrentTransformerRatio:= uiCurrentTransformerRatio_EM0, 
	nSlaveAddr 	:= 1001,
	stEL3443_IO := ,
	pDpmData=> , 
	stDataEMPower=> , 
	stDataEMCounter=> , 
	stDataEMPowerRealTime=> , 
	stDataEMCounterRealTime=> );

fb_EL3443_EM0.stEL3443_IO.MDP5001_341_Input := stEL3443_IO_1.MDP5001_341_Input;
stEL3443_IO_1.MDP5001_341_Output	:= fb_EL3443_EM0.stEL3443_IO.MDP5001_341_Output;
 	
lr_RealPower_EM0 			:= fb_EL3443_EM0.stDataEMPower.lrPowerTotal; 	
lr_ApparentPower_EM0 		:= fb_EL3443_EM0.stDataEMPower.lrApparentPowerTotal;
lr_ReactivePower_EM0		:= fb_EL3443_EM0.stDataEMPower.lrReactivePowerTotal;
lr_Frequency_EM0			:= fb_EL3443_EM0.stDataEMPower.lrFrequency;
lr_Voltage_EM0_L1N			:= fb_EL3443_EM0.stDataEMPower.lrVoltageL1N;
lr_Voltage_EM0_L2N			:= fb_EL3443_EM0.stDataEMPower.lrVoltageL2N;
lr_Voltage_EM0_L3N			:= fb_EL3443_EM0.stDataEMPower.lrVoltageL3N;
lr_Voltage_EM0_L1L2			:= fb_EL3443_EM0.stDataEMPower.lrVoltageL1L2;
lr_Voltage_EM0_L2L3			:= fb_EL3443_EM0.stDataEMPower.lrVoltageL2L3;
lr_Voltage_EM0_L3L1			:= fb_EL3443_EM0.stDataEMPower.lrVoltageL3L1;
lr_EnergyCounter_EM0		:= fb_EL3443_EM0.stDataEMCounter.lrTotalCounterEnergy_Consumption;
lr_Current_EM0_L1			:= fb_EL3443_EM0.stDataEMPower.lrCurrentL1;
lr_Current_EM0_L2			:= fb_EL3443_EM0.stDataEMPower.lrCurrentL2;
lr_Current_EM0_L3			:= fb_EL3443_EM0.stDataEMPower.lrCurrentL3;


//EM1 (for single Phase Measurements, EL3446-1)
fb_EL3446_1(
	bEnable:= TRUE , 
	bEnableVariantValues:= TRUE, 
	pDpmData:= fb_EL3443_EM0.pDpmData, 
	nSlaveAddr:= 1002, 
	bInvers_CH1:= b_Invers_EM1_1, 
	bInvers_CH2:= b_Invers_EM1_2, 
	bInvers_CH3:= b_Invers_EM1_3, 
	bInvers_CH4:= b_Invers_EM1_4, 
	bInvers_CH5:= b_Invers_EM1_5, 
	bInvers_CH6:= b_Invers_EM1_6, 
	uiCurrentTransformerRatio_CH1:= uiCurrentTransformerRatio_EM1_1, 
	uiCurrentTransformerRatio_CH2:= uiCurrentTransformerRatio_EM1_2, 
	uiCurrentTransformerRatio_CH3:= uiCurrentTransformerRatio_EM1_3, 
	uiCurrentTransformerRatio_CH4:= uiCurrentTransformerRatio_EM1_4, 
	uiCurrentTransformerRatio_CH5:= uiCurrentTransformerRatio_EM1_5, 
	uiCurrentTransformerRatio_CH6:= uiCurrentTransformerRatio_EM1_6, 
	uiVoltagePhaseSelector_CH1:= ui_PhaseSelector_EM1_1, 
	uiVoltagePhaseSelector_CH2:= ui_PhaseSelector_EM1_2, 
	uiVoltagePhaseSelector_CH3:= ui_PhaseSelector_EM1_3, 
	uiVoltagePhaseSelector_CH4:= ui_PhaseSelector_EM1_4, 
	uiVoltagePhaseSelector_CH5:= ui_PhaseSelector_EM1_5, 
	uiVoltagePhaseSelector_CH6:= ui_PhaseSelector_EM1_6, 
	bEnable3PhaseCH13:= FALSE, 
	bEnable3PhaseCH46:= FALSE, 
	stDataEMPowerRealTime:= fb_EL3443_EM0.stDataEMPowerRealTime, 
	stEL3446_IO := ,
	stDataEMPower_CH1=> , 
	stDataEMCounter_CH1=> , 
	stDataEMPowerRealTime_CH1=> , 
	stDataEMCounterRealTime_CH1=> , 
	stDataEMPower_CH2=> , 
	stDataEMCounter_CH2=> , 
	stDataEMPowerRealTime_CH2=> , 
	stDataEMCounterRealTime_CH2=> , 
	stDataEMPower_CH3=> , 
	stDataEMCounter_CH3=> , 
	stDataEMPowerRealTime_CH3=> , 
	stDataEMCounterRealTime_CH3=> , 
	stDataEMPower_CH4=> , 
	stDataEMCounter_CH4=> , 
	stDataEMPowerRealTime_CH4=> , 
	stDataEMCounterRealTime_CH4=> , 
	stDataEMPower_CH5=> , 
	stDataEMCounter_CH5=> , 
	stDataEMPowerRealTime_CH5=> , 
	stDataEMCounterRealTime_CH5=> , 
	stDataEMPower_CH6=> , 
	stDataEMCounter_CH6=> , 
	stDataEMPowerRealTime_CH6=> , 
	stDataEMCounterRealTime_CH6=> );
fb_EL3446_1.stEL3446_IO.MDP5001_342_Input := stEL3446_IO_1.MDP5001_342_Input;
stEL3446_IO_1.MDP5001_342_Output := 	fb_EL3446_1.stEL3446_IO.MDP5001_342_Output;

lrPower_EM1_1				:= 	LIMIT(0,fb_EL3446_1.stDataEMPower_CH1.lrPowerTotal,1000);
lrPower_EM1_2				:= 	LIMIT(0,fb_EL3446_1.stDataEMPower_CH2.lrPowerTotal,1000);
lrPower_EM1_3				:= 	LIMIT(0,fb_EL3446_1.stDataEMPower_CH3.lrPowerTotal,1000);
lrPower_EM1_4				:= 	LIMIT(0,fb_EL3446_1.stDataEMPower_CH4.lrPowerTotal,1000);
lrPower_EM1_5				:= 	LIMIT(0,fb_EL3446_1.stDataEMPower_CH5.lrPowerTotal,1000);
lrPower_EM1_6				:= 	LIMIT(0,fb_EL3446_1.stDataEMPower_CH6.lrPowerTotal,1000);

lrPower_EM1_3p1 			:= lrPower_EM1_1 + lrPower_EM1_2 + lrPower_EM1_3;
lrPower_EM1_3p2 			:= lrPower_EM1_4 + lrPower_EM1_5 + lrPower_EM1_6;

//EM2 (for single Phase Measurements, EL3446-2)
fb_EL3446_2(
	bEnable:= TRUE , 
	bEnableVariantValues:= TRUE, 
	pDpmData:= fb_EL3443_EM0.pDpmData, 
	nSlaveAddr:= 1003, 
	bInvers_CH1:= b_Invers_EM2_1, 
	bInvers_CH2:= b_Invers_EM2_2, 
	bInvers_CH3:= b_Invers_EM2_3, 
	bInvers_CH4:= b_Invers_EM2_4, 
	bInvers_CH5:= b_Invers_EM2_5, 
	bInvers_CH6:= b_Invers_EM2_6, 
	uiCurrentTransformerRatio_CH1:= uiCurrentTransformerRatio_EM2_1, 
	uiCurrentTransformerRatio_CH2:= uiCurrentTransformerRatio_EM2_2, 
	uiCurrentTransformerRatio_CH3:= uiCurrentTransformerRatio_EM2_3, 
	uiCurrentTransformerRatio_CH4:= uiCurrentTransformerRatio_EM2_4, 
	uiCurrentTransformerRatio_CH5:= uiCurrentTransformerRatio_EM2_5, 
	uiCurrentTransformerRatio_CH6:= uiCurrentTransformerRatio_EM2_6, 
	uiVoltagePhaseSelector_CH1:= ui_PhaseSelector_EM2_1, 
	uiVoltagePhaseSelector_CH2:= ui_PhaseSelector_EM2_2, 
	uiVoltagePhaseSelector_CH3:= ui_PhaseSelector_EM2_3, 
	uiVoltagePhaseSelector_CH4:= ui_PhaseSelector_EM2_4, 
	uiVoltagePhaseSelector_CH5:= ui_PhaseSelector_EM2_5, 
	uiVoltagePhaseSelector_CH6:= ui_PhaseSelector_EM2_6, 
	bEnable3PhaseCH13:= FALSE, 
	bEnable3PhaseCH46:= FALSE, 
	stDataEMPowerRealTime:= fb_EL3443_EM0.stDataEMPowerRealTime, 
	stEL3446_IO := ,
	stDataEMPower_CH1=> , 
	stDataEMCounter_CH1=> , 
	stDataEMPowerRealTime_CH1=> , 
	stDataEMCounterRealTime_CH1=> , 
	stDataEMPower_CH2=> , 
	stDataEMCounter_CH2=> , 
	stDataEMPowerRealTime_CH2=> , 
	stDataEMCounterRealTime_CH2=> , 
	stDataEMPower_CH3=> , 
	stDataEMCounter_CH3=> , 
	stDataEMPowerRealTime_CH3=> , 
	stDataEMCounterRealTime_CH3=> , 
	stDataEMPower_CH4=> , 
	stDataEMCounter_CH4=> , 
	stDataEMPowerRealTime_CH4=> , 
	stDataEMCounterRealTime_CH4=> , 
	stDataEMPower_CH5=> , 
	stDataEMCounter_CH5=> , 
	stDataEMPowerRealTime_CH5=> , 
	stDataEMCounterRealTime_CH5=> , 
	stDataEMPower_CH6=> , 
	stDataEMCounter_CH6=> , 
	stDataEMPowerRealTime_CH6=> , 
	stDataEMCounterRealTime_CH6=> );
fb_EL3446_2.stEL3446_IO.MDP5001_342_Input := stEL3446_IO_2.MDP5001_342_Input;
stEL3446_IO_2.MDP5001_342_Output := 	fb_EL3446_2.stEL3446_IO.MDP5001_342_Output;

lrPower_EM2_1				:= 	LIMIT(0,fb_EL3446_2.stDataEMPower_CH1.lrPowerTotal,1000);
lrPower_EM2_2				:= 	LIMIT(0,fb_EL3446_2.stDataEMPower_CH2.lrPowerTotal,1000);
lrPower_EM2_3				:= 	LIMIT(0,fb_EL3446_2.stDataEMPower_CH3.lrPowerTotal,1000);
lrPower_EM2_4				:= 	LIMIT(0,fb_EL3446_2.stDataEMPower_CH4.lrPowerTotal,1000);
lrPower_EM2_5				:= 	LIMIT(0,fb_EL3446_2.stDataEMPower_CH5.lrPowerTotal,1000);
lrPower_EM2_6				:= 	LIMIT(0,fb_EL3446_2.stDataEMPower_CH6.lrPowerTotal,1000);

lrPower_EM2_3p1 			:= lrPower_EM2_1 + lrPower_EM2_2 + lrPower_EM2_3;
lrPower_EM2_3p2 			:= lrPower_EM2_4 + lrPower_EM2_5 + lrPower_EM2_6;

(*
lr_EnergyCounter_EM1	:= 	fb_EL3446_1.stDataEMCounter_CH1.lrTotalCounterEnergy_Consumption;
lr_EnergyCounter_EM2	:= 	fb_EL3446_1.stDataEMCounter_CH2.lrTotalCounterEnergy_Consumption;
lr_EnergyCounter_EM3	:= 	fb_EL3446_1.stDataEMCounter_CH3.lrTotalCounterEnergy_Consumption;
lr_EnergyCounter_EM4	:= 	fb_EL3446_1.stDataEMCounter_CH4.lrTotalCounterEnergy_Consumption;
lr_EnergyCounter_EM5	:= 	fb_EL3446_1.stDataEMCounter_CH5.lrTotalCounterEnergy_Consumption;
lr_EnergyCounter_EM6	:= 	fb_EL3446_1.stDataEMCounter_CH6.lrTotalCounterEnergy_Consumption;
*)

//EM3 (for single Phase Measurements, EL3446-3)
fb_EL3446_3(
	bEnable:= TRUE , 
	bEnableVariantValues:= TRUE, 
	pDpmData:= fb_EL3443_EM0.pDpmData, 
	nSlaveAddr:= 1004, 
	bInvers_CH1:= b_Invers_EM3_1, 
	bInvers_CH2:= b_Invers_EM3_2, 
	bInvers_CH3:= b_Invers_EM3_3, 
	bInvers_CH4:= b_Invers_EM3_4, 
	bInvers_CH5:= b_Invers_EM3_5, 
	bInvers_CH6:= b_Invers_EM3_6, 
	uiCurrentTransformerRatio_CH1:= uiCurrentTransformerRatio_EM3_1, 
	uiCurrentTransformerRatio_CH2:= uiCurrentTransformerRatio_EM3_2, 
	uiCurrentTransformerRatio_CH3:= uiCurrentTransformerRatio_EM3_3, 
	uiCurrentTransformerRatio_CH4:= uiCurrentTransformerRatio_EM3_4, 
	uiCurrentTransformerRatio_CH5:= uiCurrentTransformerRatio_EM3_5, 
	uiCurrentTransformerRatio_CH6:= uiCurrentTransformerRatio_EM3_6, 
	uiVoltagePhaseSelector_CH1:= ui_PhaseSelector_EM3_1, 
	uiVoltagePhaseSelector_CH2:= ui_PhaseSelector_EM3_2, 
	uiVoltagePhaseSelector_CH3:= ui_PhaseSelector_EM3_3, 
	uiVoltagePhaseSelector_CH4:= ui_PhaseSelector_EM3_4, 
	uiVoltagePhaseSelector_CH5:= ui_PhaseSelector_EM3_5, 
	uiVoltagePhaseSelector_CH6:= ui_PhaseSelector_EM3_6, 
	bEnable3PhaseCH13:= FALSE, 
	bEnable3PhaseCH46:= FALSE, 
	stDataEMPowerRealTime:= fb_EL3443_EM0.stDataEMPowerRealTime, 
	stEL3446_IO := ,
	stDataEMPower_CH1=> , 
	stDataEMCounter_CH1=> , 
	stDataEMPowerRealTime_CH1=> , 
	stDataEMCounterRealTime_CH1=> , 
	stDataEMPower_CH2=> , 
	stDataEMCounter_CH2=> , 
	stDataEMPowerRealTime_CH2=> , 
	stDataEMCounterRealTime_CH2=> , 
	stDataEMPower_CH3=> , 
	stDataEMCounter_CH3=> , 
	stDataEMPowerRealTime_CH3=> , 
	stDataEMCounterRealTime_CH3=> , 
	stDataEMPower_CH4=> , 
	stDataEMCounter_CH4=> , 
	stDataEMPowerRealTime_CH4=> , 
	stDataEMCounterRealTime_CH4=> , 
	stDataEMPower_CH5=> , 
	stDataEMCounter_CH5=> , 
	stDataEMPowerRealTime_CH5=> , 
	stDataEMCounterRealTime_CH5=> , 
	stDataEMPower_CH6=> , 
	stDataEMCounter_CH6=> , 
	stDataEMPowerRealTime_CH6=> , 
	stDataEMCounterRealTime_CH6=> );
fb_EL3446_3.stEL3446_IO.MDP5001_342_Input := stEL3446_IO_3.MDP5001_342_Input;
stEL3446_IO_3.MDP5001_342_Output := 	fb_EL3446_3.stEL3446_IO.MDP5001_342_Output;

lrPower_EM3_1				:= 	LIMIT(0,fb_EL3446_3.stDataEMPower_CH1.lrPowerTotal,1000);
lrPower_EM3_2				:= 	LIMIT(0,fb_EL3446_3.stDataEMPower_CH2.lrPowerTotal,1000);
lrPower_EM3_3				:= 	LIMIT(0,fb_EL3446_3.stDataEMPower_CH3.lrPowerTotal,1000);
lrPower_EM3_4				:= 	LIMIT(0,fb_EL3446_3.stDataEMPower_CH4.lrPowerTotal,1000);
lrPower_EM3_5				:= 	LIMIT(0,fb_EL3446_3.stDataEMPower_CH5.lrPowerTotal,1000);
lrPower_EM3_6				:= 	LIMIT(0,fb_EL3446_3.stDataEMPower_CH6.lrPowerTotal,1000);

lrPower_EM3_3p1 			:= lrPower_EM3_1 + lrPower_EM3_2 + lrPower_EM3_3;
lrPower_EM3_3p2 			:= lrPower_EM3_4 + lrPower_EM3_5 + lrPower_EM3_6;


//EM4 (for single Phase Measurements, EL3446-4)
fb_EL3446_4(
	bEnable:= TRUE , 
	bEnableVariantValues:= TRUE, 
	pDpmData:= fb_EL3443_EM0.pDpmData, 
	nSlaveAddr:= 1005, 
	bInvers_CH1:= b_Invers_EM4_1, 
	bInvers_CH2:= b_Invers_EM4_2, 
	bInvers_CH3:= b_Invers_EM4_3, 
	bInvers_CH4:= b_Invers_EM4_4, 
	bInvers_CH5:= b_Invers_EM4_5, 
	bInvers_CH6:= b_Invers_EM4_6, 
	uiCurrentTransformerRatio_CH1:= uiCurrentTransformerRatio_EM4_1, 
	uiCurrentTransformerRatio_CH2:= uiCurrentTransformerRatio_EM4_2, 
	uiCurrentTransformerRatio_CH3:= uiCurrentTransformerRatio_EM4_3, 
	uiCurrentTransformerRatio_CH4:= uiCurrentTransformerRatio_EM4_4, 
	uiCurrentTransformerRatio_CH5:= uiCurrentTransformerRatio_EM4_5, 
	uiCurrentTransformerRatio_CH6:= uiCurrentTransformerRatio_EM4_6, 
	uiVoltagePhaseSelector_CH1:= ui_PhaseSelector_EM4_1, 
	uiVoltagePhaseSelector_CH2:= ui_PhaseSelector_EM4_2, 
	uiVoltagePhaseSelector_CH3:= ui_PhaseSelector_EM4_3, 
	uiVoltagePhaseSelector_CH4:= ui_PhaseSelector_EM4_4, 
	uiVoltagePhaseSelector_CH5:= ui_PhaseSelector_EM4_5, 
	uiVoltagePhaseSelector_CH6:= ui_PhaseSelector_EM4_6, 
	bEnable3PhaseCH13:= FALSE, 
	bEnable3PhaseCH46:= FALSE, 
	stDataEMPowerRealTime:= fb_EL3443_EM0.stDataEMPowerRealTime, 
	stEL3446_IO := ,
	stDataEMPower_CH1=> , 
	stDataEMCounter_CH1=> , 
	stDataEMPowerRealTime_CH1=> , 
	stDataEMCounterRealTime_CH1=> , 
	stDataEMPower_CH2=> , 
	stDataEMCounter_CH2=> , 
	stDataEMPowerRealTime_CH2=> , 
	stDataEMCounterRealTime_CH2=> , 
	stDataEMPower_CH3=> , 
	stDataEMCounter_CH3=> , 
	stDataEMPowerRealTime_CH3=> , 
	stDataEMCounterRealTime_CH3=> , 
	stDataEMPower_CH4=> , 
	stDataEMCounter_CH4=> , 
	stDataEMPowerRealTime_CH4=> , 
	stDataEMCounterRealTime_CH4=> , 
	stDataEMPower_CH5=> , 
	stDataEMCounter_CH5=> , 
	stDataEMPowerRealTime_CH5=> , 
	stDataEMCounterRealTime_CH5=> , 
	stDataEMPower_CH6=> , 
	stDataEMCounter_CH6=> , 
	stDataEMPowerRealTime_CH6=> , 
	stDataEMCounterRealTime_CH6=> );
fb_EL3446_4.stEL3446_IO.MDP5001_342_Input := stEL3446_IO_4.MDP5001_342_Input;
stEL3446_IO_4.MDP5001_342_Output := 	fb_EL3446_4.stEL3446_IO.MDP5001_342_Output;

lrPower_EM4_1				:= 	LIMIT(0,fb_EL3446_4.stDataEMPower_CH1.lrPowerTotal,1000);
lrPower_EM4_2				:= 	LIMIT(0,fb_EL3446_4.stDataEMPower_CH2.lrPowerTotal,1000);
lrPower_EM4_3				:= 	LIMIT(0,fb_EL3446_4.stDataEMPower_CH3.lrPowerTotal,1000);
lrPower_EM4_4				:= 	LIMIT(0,fb_EL3446_4.stDataEMPower_CH4.lrPowerTotal,1000);
lrPower_EM4_5				:= 	LIMIT(0,fb_EL3446_4.stDataEMPower_CH5.lrPowerTotal,1000);
lrPower_EM4_6				:= 	LIMIT(0,fb_EL3446_4.stDataEMPower_CH6.lrPowerTotal,1000);

lrPower_EM4_3p1 			:= lrPower_EM4_1 + lrPower_EM4_2 + lrPower_EM4_3;
lrPower_EM4_3p2 			:= lrPower_EM4_4 + lrPower_EM4_5 + lrPower_EM4_6;

END_PROGRAM

// ---- POUs/prgTmp.TcPOU
PROGRAM prgTmp
VAR
	fbPT100Reader : FB_PT100_Read;
    pt100_Channel1 : REAL;           								// Variablen für den PT100-Wert
    pt100_Channel2 : REAL;           
    temperature1 : REAL;            								//{#lynus.ag#()}
    temperature2 : REAL;        									//{#lynus.ag#()}
	{attribute 'TcLinkTo' := 'TIID^Device 2 (EtherCAT)^Term 1 (EK1200)^Term 7 (EL3202)^RTD Inputs Channel 1^Value'}
	EL3202_Channel_1 AT%I*: INT;
	{attribute 'TcLinkTo' := 'TIID^Device 2 (EtherCAT)^Term 1 (EK1200)^Term 7 (EL3202)^RTD Inputs Channel 2^Value'}
	EL3202_Channel_2 AT%I*: INT;
END_VAR

fbPT100Reader(
				EL3202_Channel_1 := EL3202_Channel_1, 
				EL3202_Channel_2 := EL3202_Channel_2, 
				bScale := TRUE);
				
temperature1 := fbPT100Reader.temperature1;
temperature2 := fbPT100Reader.temperature2;

END_PROGRAM

// ---- FBs/FB_PT100_Read.TcPOU
FUNCTION_BLOCK FB_PT100_Read
VAR_INPUT
    bScale : BOOL := TRUE;
    EL3202_Channel_1: INT;  
    EL3202_Channel_2: INT;  
END_VAR
VAR_OUTPUT
    temperature1 : REAL;   // Berechnete Temperatur
    temperature2 : REAL;   
END_VAR

IF bScale THEN
	temperature1 := TO_REAL(EL3202_Channel_1) / 10;
	temperature2 := TO_REAL(EL3202_Channel_2) / 10;
END_IF

END_FUNCTION_BLOCK

// ---- POUs/prgComEffIO.TcPOU
PROGRAM prgComEffIO
VAR
	fbCom		: FB_MqttCommunicator_V5;
	int_SSPNumber: INT;
END_VAR

fbCom(
	bConnect:= TRUE, 
	strAuthKey:= 'ENE87365342998', 
	sUserName:= , 
	sUserPassword:= , 
	eSavePositionCertificate:= eSavePositionOnPLC.ePostionHardDisk,  
	bConnected=> , 
	bError=> , 
	hrErrorCode=> , 
	eConnectionState=> , 
	eErrorMessage_Out=> );


prg_ReadDeviceName();
IF prg_ReadDeviceName.sDeviceName = '' THEN
	prg_ReadDeviceName.bStart := TRUE;
END_IF


// select user / pass according device name:

IF prg_ReadDeviceName.sDeviceName = 'EIOSM000002' THEN
	fbCom.sUserName:= '0b42849c-4998-452d-bcd9-1344b044b06a'; 
    fbCom.sUserPassword:= '8be448ae-72bb-402a-8881-f106399ccc0a';
	int_SSPNumber :=2;
ELSIF prg_ReadDeviceName.sDeviceName = 'EIOSM000003' THEN
	fbCom.sUserName:= '250c21dc-16ee-4d4b-a8b6-b80fa572657e'; 
    fbCom.sUserPassword:= '131f7038-8c5a-467b-8f48-3b98e46b3e9d';
	int_SSPNumber :=3;
ELSIF prg_ReadDeviceName.sDeviceName = 'EIOSM000004' THEN
	fbCom.sUserName:= 'c938aafa-9a8d-47b6-9d90-e88759d88525'; 
    fbCom.sUserPassword:= '03531b94-b497-4a3f-9018-b2efc52058ad';
	int_SSPNumber :=4;
ELSIF prg_ReadDeviceName.sDeviceName = 'EIOSM000001' THEN
	fbCom.sUserName:= 'c5a26c3c-d7be-49fa-bb4b-d09878f078e1'; 
    fbCom.sUserPassword:= '835df6a6-a36a-4edd-98fd-f6a495ce7360';
	int_SSPNumber :=1;
END_IF

END_PROGRAM
